// TIA Portal V20 export
DATA_BLOCK "CallUnit_DB"   // DB147
// stored: AssignedProDiagFB Unit1.ProDiag, InstanceOfName Unit1.CallUnit, InstanceOfType FB, Namespace Unit1
"Unit1.CallUnit"
   // VAR_INPUT
   //    safetyReleased : Bool;
   // END_VAR
   // VAR_OUTPUT
   //    acknowledgeSafety { ExternalWritable := 'False'} : Bool;
   // END_VAR
   // VAR_IN_OUT
   //    globalStatus : "LAF_typeGeneralStatus";
   //    unitInterface : "LAF_typeUnitInterface";
   // END_VAR
   // VAR
   //    instManageAlarms { ExternalWritable := 'False'} : "LAF_ManageAlarms";
   //    instStatusCollector { ExternalWritable := 'False'} : "LUC_StatusCollector";
   //    instInterfaceManager { ExternalWritable := 'False'} : "LUC_InterfaceManager";
   //    instUnitModeStateManager { ExternalWritable := 'False'} : "LPMLV2022_UnitModeStateManager";
   //    instRemoteInterfaceOpcUa { ExternalWritable := 'False'} : "LUC_RemoteCtrl_OpcUa";
   //    instSignalStack { ExternalWritable := 'False'} : "LUC_SignalStack";
   //    instUnitModeStateTimes { ExternalWritable := 'False'} : "LPMLV2022_UnitModeStateTimes";
   //    instUnitModeChangeAllowed { ExternalWritable := 'False'} : "LPMLV2022_UnitModeChangeAllowed";
   //    instPFEEvents { ExternalWritable := 'False'} : "Unit1.EventsPFE";
   //    instTonTimer { ExternalWritable := 'False'} : Array[0..9] of TON_TIME;
   //    instTofTimer { ExternalWritable := 'False'} : Array[0..9] of TOF_TIME;
   //    instEQP_Interface_BA030 { ExternalWritable := 'False'} : "LER_EQP_Interface";
   //    instEQP_Interface_BA040 { ExternalWritable := 'False'} : "LER_EQP_Interface";
   //    instSinaInfeed { ExternalWritable := 'False'} : SinaInfeed;
   //    instLER_FFU_LIU117 { ExternalWritable := 'False'} : "LER_FFU_LIU117";
   //    statRemoteInterface { ExternalWritable := 'False'} : "LUC_typeCommands";
   //    statLocalInterface { ExternalWritable := 'False'} : "LUC_typeCommands";
   //    statEmEnableCheck { ExternalWritable := 'False'} : Array[0..2] of Bool;
   //    statEmHomedCheck { ExternalWritable := 'False'} : Array[0..2] of Bool;
   //    statPulse { ExternalWritable := 'False'} : Array[0..99] of Bool;
   //    statCycleTime { ExternalWritable := 'False'} : Struct
   //       Buffer1 : LReal;
   //       Buffer2 : DInt;
   //       Buffer3 : DInt;
   //       Buffer4 : DInt;
   //       Buffer5 : DInt;
   //    END_STRUCT;
   //    statEnableManualCmds : Bool;
   //    statAllEmLinked { ExternalWritable := 'False'} : Bool;
   //    citi_Ptrig : Array[0..20] of Bool;
   //    citiTon : Array[0..20] of TON_TIME;
   //    citi : Time;
   //    citiTest : Array[0..20] of Bool;
   // END_VAR
BEGIN
END_DATA_BLOCK
